FUNCTION IsValidOutputPort : BOOL
VAR_INPUT
	OutputPort : I_OutputPort;
END_VAR

IsValidOutputPort := OutputPort <> 0;

END_FUNCTION

(* stored: Version 1.1.0.1, ProductVersion 3.1.4024.12
   POU IsValidOutputPort: Id {9449dc11-2905-0e27-09f9-d6c303c2e5af}, SpecialFunc None *)
